Universal Robots PolyScope program: examen_e8.urp

Program examen_e8 (installation=default directory=/home/hugo/Documents/Proyecto_Ingenieria/ursim-5.10.2.106319/programs/ASM/Clase4_ActividadPractica createdIn=5.9.4.1031232 lastSavedIn=5.10.2.106319 robotSerialNumber=20195599999)
Calibrated DH parameters: a=[0, -0.425, -0.3922, 0, 0, 0]; d=[0.1625, 0, 0, 0.1333, 0.0997, 0.0996]; alpha=[1.570796, 0, 0, 1.570796, -1.570796, 0]; deltaTheta=[0, 0, 0, 0, 0, 0]
Robot Program (runOnlyOnce=true)
  continuar :=  (valueSource=Operator message=¿Empezar? valueType=Boolean)
  Loop While (checkContinuously=false) expression=continuar≟ True
    Folder Estrella
      MoveL speed 250 mm/s, acceleration 1200 mm/s^2 (useActiveTCP=true) feature=Base
        Waypoint Waypoint_1 (Relative): relativeFromPosition TCP in base x=0 y=-400 z=200 mm, rx=-0.0012 ry=3.1163 rz=0.0389 rad; joints [-71.015, -91.616, -135.259, -44.011, 91.823, 18.926] deg; TCP in base x=160 y=-400 z=200 mm, rx=-0.0012 ry=3.1163 rz=0.0389 rad; joints [-50.664, -95.742, -130.97, -43.484, 92.017, 39.287] deg
        Waypoint Waypoint_4 (Relative): relativeFromPosition TCP in base x=0 y=-400 z=200 mm, rx=-0.0012 ry=3.1163 rz=0.0389 rad; joints [-71.015, -91.616, -135.259, -44.011, 91.823, 18.926] deg; TCP in base x=-129.44 y=-400 z=105.95 mm, rx=-0.0012 ry=3.1163 rz=0.0389 rad; joints [-89.806, -109.02, -136.284, -26.122, 91.441, 0.131] deg
        Waypoint Waypoint_2 (Relative): relativeFromPosition TCP in base x=0 y=-400 z=200 mm, rx=-0.0012 ry=3.1163 rz=0.0389 rad; joints [-71.015, -91.616, -135.259, -44.011, 91.823, 18.926] deg; TCP in base x=49.44 y=-400 z=352.17 mm, rx=-0.0012 ry=3.1163 rz=0.0389 rad; joints [-64.142, -77.956, -120.673, -72.032, 91.916, 25.802] deg
        Waypoint Waypoint_5 (Relative): relativeFromPosition TCP in base x=0 y=-400 z=200 mm, rx=-0.0012 ry=3.1163 rz=0.0389 rad; joints [-71.015, -91.616, -135.259, -44.011, 91.823, 18.926] deg; TCP in base x=49.44 y=-400 z=47.84 mm, rx=-0.0012 ry=3.1163 rz=0.0389 rad; joints [-64.142, -119.225, -139.681, -11.755, 91.916, 25.802] deg
        Waypoint Waypoint_3 (Relative): relativeFromPosition TCP in base x=0 y=-400 z=200 mm, rx=-0.0012 ry=3.1163 rz=0.0389 rad; joints [-71.015, -91.616, -135.259, -44.011, 91.823, 18.926] deg; TCP in base x=-129.44 y=-400 z=294 mm, rx=-0.0012 ry=3.1163 rz=0.0389 rad; joints [-89.806, -84.462, -124.43, -62.534, 91.441, 0.131] deg
        Waypoint Waypoint_1 (Relative): relativeFromPosition TCP in base x=0 y=-400 z=200 mm, rx=-0.0012 ry=3.1163 rz=0.0389 rad; joints [-71.015, -91.616, -135.259, -44.011, 91.823, 18.926] deg; TCP in base x=160 y=-400 z=200 mm, rx=-0.0012 ry=3.1163 rz=0.0389 rad; joints [-50.664, -95.742, -130.97, -43.484, 92.017, 39.287] deg
    continuar :=  (valueSource=Operator message=¿Continuar? valueType=Boolean)
